// Mitsubishi GX Works2 project: limit   PLC: FX3U/FX3UC

PROGRAM MAIN
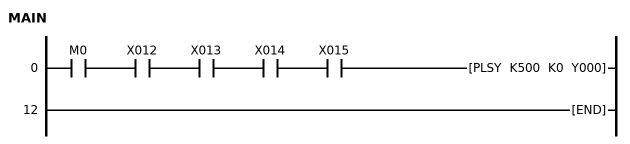
0     LD      M0
      AND     X012
      AND     X013
      AND     X014
      AND     X015
      PLSY    K500 K0 Y000
12    END
END_PROGRAM
